FUNCTION_BLOCK E_MERGE7
  (* Version 1.0, 2005-09-22, Goran Cengic, Chalmers *)
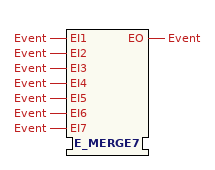
  EVENT_INPUT
    EI1;
    EI2;
    EI3;
    EI4;
    EI5;
    EI6;
    EI7;
  END_EVENT
  EVENT_OUTPUT
    EO;
  END_EVENT
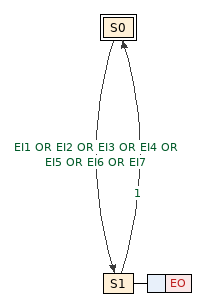
  EC_STATES
    S0;
    S1 : -> EO;
  END_STATES
  EC_TRANSITIONS
    S0 TO S1 := EI1 OR EI2 OR EI3 OR EI4 OR EI5 OR EI6 OR EI7;
    S1 TO S0 := 1;
  END_TRANSITIONS
END_FUNCTION_BLOCK
